(* PLC project Unnamed, Unknown Unnamed 1 *)
(* stored: creationDateTime 2024-06-09T17:07:02, modificationDateTime 2024-06-10T06:26:47 *)

PROGRAM Stoplight
  VAR
    redEW AT %QX0.3 : BOOL;
    redEW0 AT %QX0.4 : BOOL;
    yellEW AT %QX0.2 : BOOL;
    greenEWLight AT %QW2 : UINT;
    yellNS AT %QX0.1 : BOOL;
    greenNS AT %QX0.0 : BOOL;
    redNSLight AT %QW0 : UINT;
  END_VAR
  VAR
    redNS : BOOL;
    greenEW : BOOL;
    start : BOOL;
  END_VAR
  VAR
    carEW1 AT %IX0.0 : BOOL;
    carEW2 AT %IX0.1 : BOOL;
  END_VAR
  VAR
    TP0 : TP;
    TP1 : TP;
    TP2 : TP;
    TP3 : TP;
    TP4 : TP;
    TP5 : TP;
    TON0 : TON;
    TON1 : TON;
  END_VAR
  VAR  (* added by the conversion: wires and edge detectors of the diagram *)
    F_TRIG1 : F_TRIG;
    F_TRIG2 : F_TRIG;
    R_TRIG3 : R_TRIG;
    F_TRIG4 : F_TRIG;
    F_TRIG5 : F_TRIG;
  END_VAR

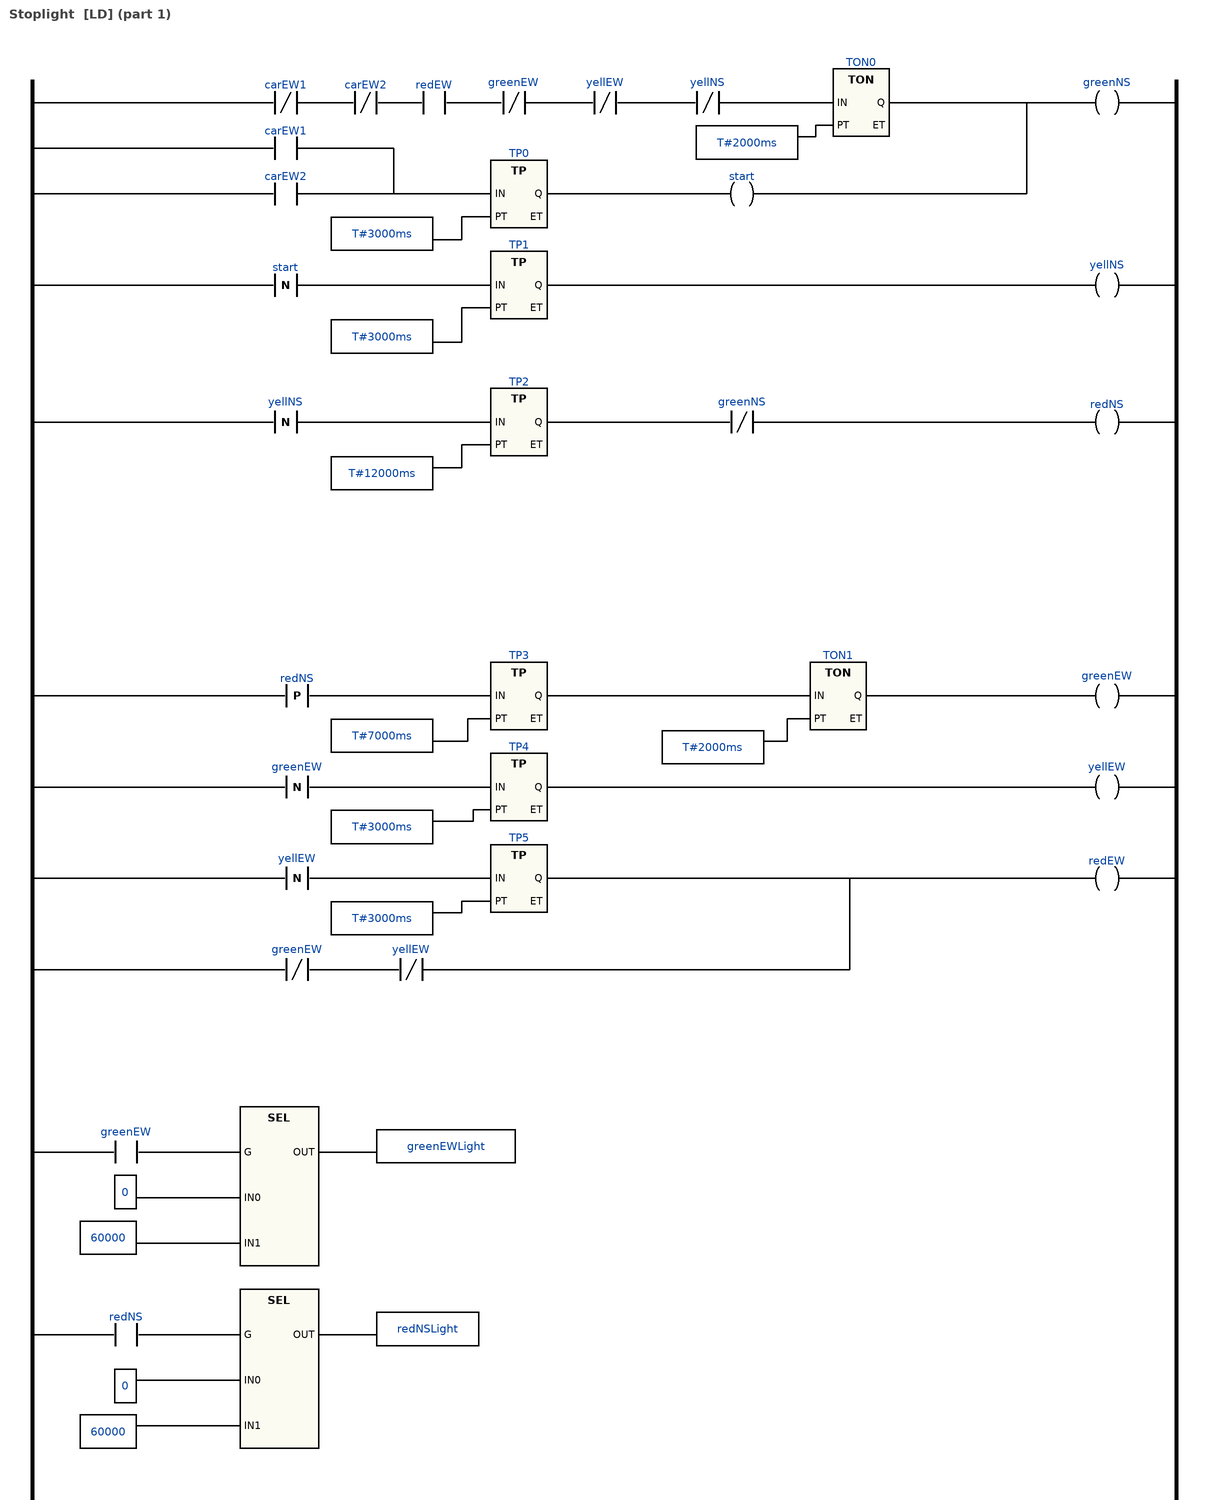
(* LD diagram, written out as Structured Text *)
greenEWLight := SEL(greenEW, 0, 60000);
redNSLight := SEL(redNS, 0, 60000);
TP0(IN := carEW1 OR carEW2, PT := T#3000ms);
TON0(IN := NOT carEW1 AND NOT carEW2 AND redEW AND NOT greenEW AND NOT yellEW AND NOT yellNS, PT := T#2000ms);
greenNS := TP0.Q OR TON0.Q;
F_TRIG1(CLK := start);
TP1(IN := F_TRIG1.Q, PT := T#3000ms);
yellNS := TP1.Q;
F_TRIG2(CLK := yellNS);
TP2(IN := F_TRIG2.Q, PT := T#12000ms);
redNS := TP2.Q AND NOT greenNS;
R_TRIG3(CLK := redNS);
TP3(IN := R_TRIG3.Q, PT := T#7000ms);
TON1(IN := TP3.Q, PT := T#2000ms);
greenEW := TON1.Q;
F_TRIG4(CLK := greenEW);
TP4(IN := F_TRIG4.Q, PT := T#3000ms);
yellEW := TP4.Q;
F_TRIG5(CLK := yellEW);
TP5(IN := F_TRIG5.Q, PT := T#3000ms);
redEW := NOT greenEW AND NOT yellEW OR TP5.Q;
start := TP0.Q;
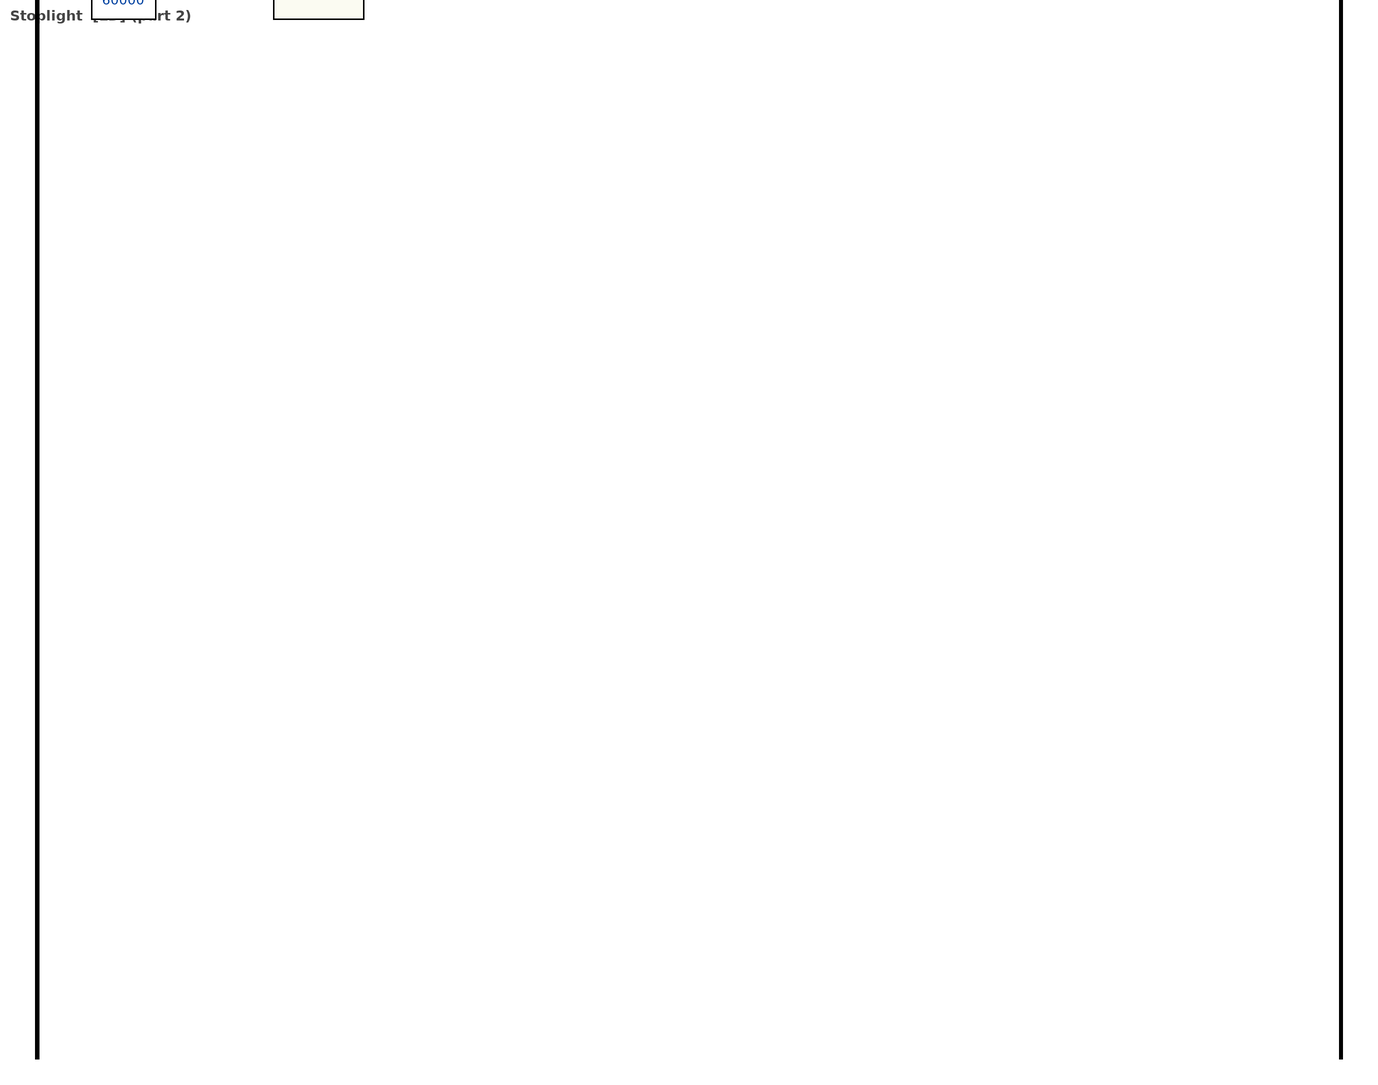
END_PROGRAM

CONFIGURATION Config0
  RESOURCE Res0 ON PLC
    TASK task0(INTERVAL := T#20ms, PRIORITY := 0);
    PROGRAM instance0 WITH task0 : Stoplight;
  END_RESOURCE
END_CONFIGURATION
